FUNCTION INTERNAL LogLevel_To_AdsLogMsgType : DWORD
VAR_INPUT
	LogLevel : E_LogLevel;
END_VAR
VAR
	retVal : DWORD; 
END_VAR

CASE LogLevel OF
	E_LogLevel.Debug, E_LogLevel.Information:
		retVal := Tc2_System.ADSLOG_MSGTYPE_HINT;
	E_LogLevel.Warning:
		retVal := Tc2_System.ADSLOG_MSGTYPE_WARN;
	E_LogLevel.Error, E_LogLevel.Fatal:
		retVal := Tc2_System.ADSLOG_MSGTYPE_ERROR;
	ELSE
		retVal := Tc2_System.ADSLOG_MSGTYPE_HINT;
END_CASE

LogLevel_To_AdsLogMsgType := retVal;

END_FUNCTION

(* stored: Version 1.1.0.1
   POU LogLevel_To_AdsLogMsgType: Id {c5255ff0-b51b-42de-ab62-e7b30a9b316a}, SpecialFunc None *)
